{attribute 'GeneratedUsingTerminal: BK1120-0000-0018'}
{attribute addProperty BoxType "BK1120-0000-0018"}
{attribute addProperty Id "Term_378_KL1002KL1002_BB38DA8F0"}
{attribute addProperty CRC "3269449944"}
{attribute addProperty Size "0"}
TYPE A_0005_BK1120_0000_0018_C2DFD8D8 EXTENDS BK1120_A2FCADE7 :
STRUCT
	{attribute addProperty Name "Term_378_KL1002"}
	Term_378_KL1002 : KL1002_BB38DA8F;
END_STRUCT
END_TYPE

(* stored: Version 1.2.0.0, ProductVersion 3.1.4024.9
   DUT A_0005_BK1120_0000_0018_C2DFD8D8: Id {93e7da85-e518-413d-a8bb-94703374f879} *)
